// Mitsubishi GX Works2 project: 5   PLC: FX3U/FX3UC

PROGRAM MAIN
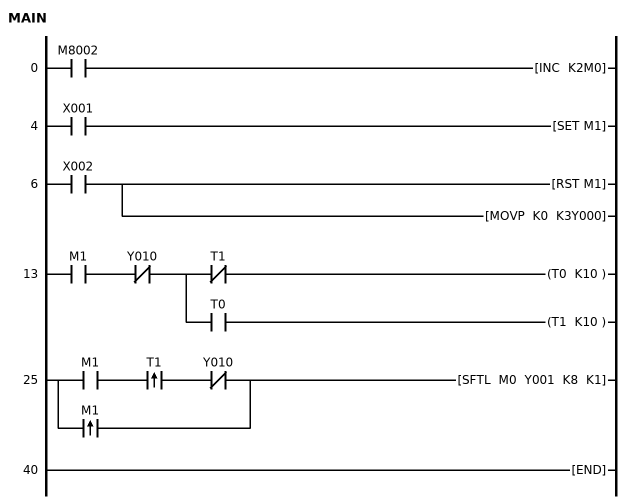
0     LD      M8002
      INC     K2M0
4     LD      X001
      SET     M1
6     LD      X002
      RST     M1
      MOVP    K0 K3Y000
13    LD      M1
      ANI     Y010
      MPS
      ANI     T1
      OUT     T0 K10
      MPP
      AND     T0
      OUT     T1 K10
25    LD      M1
      ANDP    T1
      ANI     Y010
      ORP     M1
      SFTL    M0 Y001 K8 K1
40    END
END_PROGRAM
